PROGRAM prgLynusVar
VAR
	fbVarInfo		: FB_VarInfo_V3;
	fbRW1			: FB_ReadWrite_V2;
//	fbRW2			: FB_ReadWrite;
END_VAR

fbVarInfo(
	bReadInfo:= , 
	eTMCFile:= eSelectTMCFile.eDontUseTMCFile, 
	eSavePositionTMCFile:= eSavePositionOnPLC.ePostionHardDisk, 
	udiCounterFoundVariables=> , 
	bError=> , 
	bBusy=> , 
	byProgress=> , 
	udiErrorCodeOut=> , 
	eErrorVarInfo_Out=> , 
	sVarWithError=> );
	
fbRW1(
	eUploadType:= 3 , // change and interval 5 min
	bBusy=> , 
	bError=> , 
	udiErrorCodeOut=> , 
	eErrorReadWrite_Out=> );

END_PROGRAM

(* stored: Version 1.1.0.1, ProductVersion 3.1.4024.12
   POU prgLynusVar: Id {e8e91620-bd0e-4bd4-8bb1-e4b457878fc1}, SpecialFunc None *)
